// TIA Portal V19 export
DATA_BLOCK "iDB_ScaleValueCarBodyDetection"   // DB10
{ DB_Accessible_From_OPC_UA := 'FALSE' }
// stored: AutoNumber false, DBAccessibleFromOPCUA false, DBAccessibleFromWebserver false, InstanceOfName FB_ScaleValueIntReal, InstanceOfType FB
"FB_ScaleValueIntReal"
   // VAR_INPUT
   //    xExecute { ExternalAccessible := 'False'; ExternalVisible := 'False'; ExternalWritable := 'False'} : Bool;
   //    nInputValue { ExternalAccessible := 'False'; ExternalVisible := 'False'; ExternalWritable := 'False'} : Int;
   //    stConfig { ExternalAccessible := 'False'; ExternalVisible := 'False'; ExternalWritable := 'False'} : "stConfigScaleIntReal";
   // END_VAR
   // VAR_OUTPUT
   //    stResult { ExternalAccessible := 'False'; ExternalVisible := 'False'; ExternalWritable := 'False'} : "stResult";
   //    rOutputValue { ExternalAccessible := 'False'; ExternalVisible := 'False'; ExternalWritable := 'False'} : Real;
   // END_VAR
   // VAR
   //    srNormalise { ExternalAccessible := 'False'; ExternalVisible := 'False'; ExternalWritable := 'False'} : Real;
   //    srConvertie { ExternalAccessible := 'False'; ExternalVisible := 'False'; ExternalWritable := 'False'} : Real;
   // END_VAR
BEGIN
END_DATA_BLOCK
